% RSLogix 500 project I2P Hands-On 4 - Luke.RSS, saved by version 10.00.00.00 %
PROJECT "UNTITLED"    % processor: Bul.1763 MicroLogix 1100 Series B %

PROGRAM FILES
  LAD 2   13 rungs

DATA FILES
  O0 OUTPUT  4 elements
  I1 INPUT  6 elements
  S2 STATUS  66 elements
  B3 BINARY  1 elements
  T4 TIMER  2 elements
  C5 COUNTER  1 elements
  R6 CONTROL  1 elements
  N7 INTEGER  1 elements
  F8 FLOAT  1 elements

LADDER 2
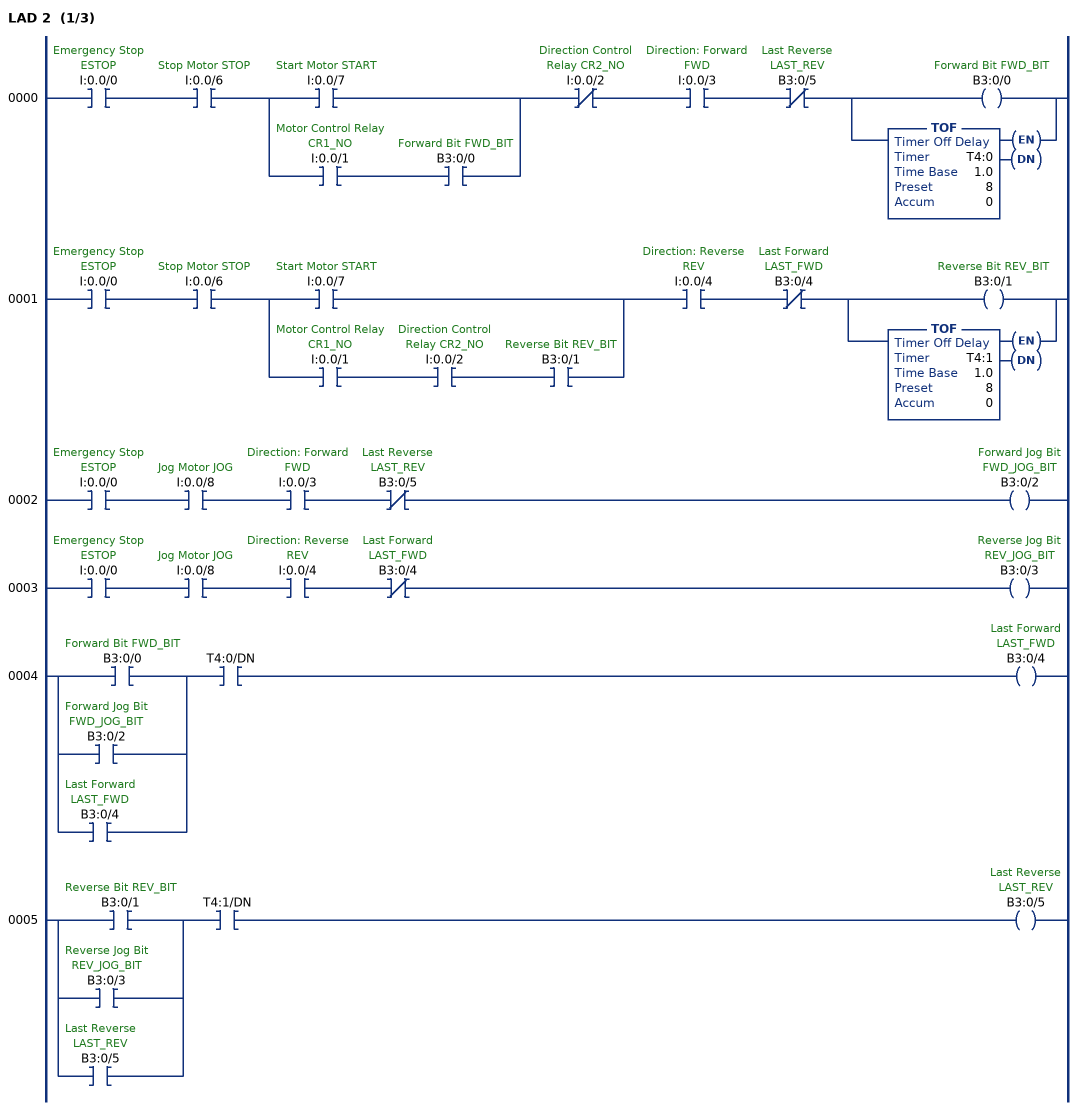
% Rung: 0 %
SOR XIC I:0.0/0 XIC I:0.0/6 BST XIC I:0.0/7 NXB XIC I:0.0/1 XIC B3:0/0 BND XIO I:0.0/2 XIC I:0.0/3 XIO B3:0/5 BST OTE B3:0/0 NXB TOF T4:0 1.0 8 0 BND EOR
%   I:0.0/0  ESTOP  "Emergency Stop" %
%   I:0.0/6  STOP  "Stop Motor" %
%   I:0.0/7  START  "Start Motor" %
%   I:0.0/1  CR1_NO  "Motor Control Relay" %
%   B3:0/0  FWD_BIT  "Forward Bit" %
%   I:0.0/2  CR2_NO  "Direction Control Relay" %
%   I:0.0/3  FWD  "Direction: Forward" %
%   B3:0/5  LAST_REV  "Last Reverse" %
% Rung: 1 %
SOR XIC I:0.0/0 XIC I:0.0/6 BST XIC I:0.0/7 NXB XIC I:0.0/1 XIC I:0.0/2 XIC B3:0/1 BND XIC I:0.0/4 XIO B3:0/4 BST OTE B3:0/1 NXB TOF T4:1 1.0 8 0 BND EOR
%   I:0.0/0  ESTOP  "Emergency Stop" %
%   I:0.0/6  STOP  "Stop Motor" %
%   I:0.0/7  START  "Start Motor" %
%   I:0.0/1  CR1_NO  "Motor Control Relay" %
%   I:0.0/2  CR2_NO  "Direction Control Relay" %
%   B3:0/1  REV_BIT  "Reverse Bit" %
%   I:0.0/4  REV  "Direction: Reverse" %
%   B3:0/4  LAST_FWD  "Last Forward" %
% Rung: 2 %
SOR XIC I:0.0/0 XIC I:0.0/8 XIC I:0.0/3 XIO B3:0/5 OTE B3:0/2 EOR
%   I:0.0/0  ESTOP  "Emergency Stop" %
%   I:0.0/8  JOG  "Jog Motor" %
%   I:0.0/3  FWD  "Direction: Forward" %
%   B3:0/5  LAST_REV  "Last Reverse" %
%   B3:0/2  FWD_JOG_BIT  "Forward Jog Bit" %
% Rung: 3 %
SOR XIC I:0.0/0 XIC I:0.0/8 XIC I:0.0/4 XIO B3:0/4 OTE B3:0/3 EOR
%   I:0.0/0  ESTOP  "Emergency Stop" %
%   I:0.0/8  JOG  "Jog Motor" %
%   I:0.0/4  REV  "Direction: Reverse" %
%   B3:0/4  LAST_FWD  "Last Forward" %
%   B3:0/3  REV_JOG_BIT  "Reverse Jog Bit" %
% Rung: 4 %
SOR BST XIC B3:0/0 NXB BST XIC B3:0/2 NXB XIC B3:0/4 BND BND XIC T4:0/DN OTE B3:0/4 EOR
%   B3:0/0  FWD_BIT  "Forward Bit" %
%   B3:0/2  FWD_JOG_BIT  "Forward Jog Bit" %
%   B3:0/4  LAST_FWD  "Last Forward" %
% Rung: 5 %
SOR BST XIC B3:0/1 NXB BST XIC B3:0/3 NXB XIC B3:0/5 BND BND XIC T4:1/DN OTE B3:0/5 EOR
%   B3:0/1  REV_BIT  "Reverse Bit" %
%   B3:0/3  REV_JOG_BIT  "Reverse Jog Bit" %
%   B3:0/5  LAST_REV  "Last Reverse" %

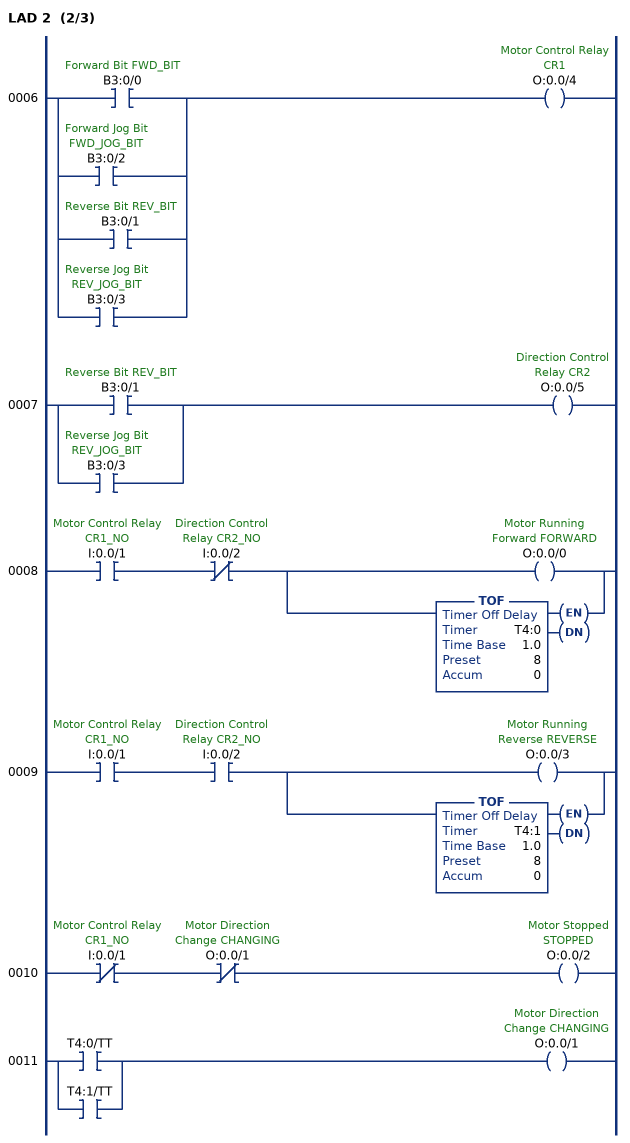
% Rung: 6 %
SOR BST XIC B3:0/0 NXB BST XIC B3:0/2 NXB BST XIC B3:0/1 NXB XIC B3:0/3 BND BND BND OTE O:0.0/4 EOR
%   B3:0/0  FWD_BIT  "Forward Bit" %
%   B3:0/2  FWD_JOG_BIT  "Forward Jog Bit" %
%   B3:0/1  REV_BIT  "Reverse Bit" %
%   B3:0/3  REV_JOG_BIT  "Reverse Jog Bit" %
%   O:0.0/4  CR1  "Motor Control Relay" %
% Rung: 7 %
SOR BST XIC B3:0/1 NXB XIC B3:0/3 BND OTE O:0.0/5 EOR
%   B3:0/1  REV_BIT  "Reverse Bit" %
%   B3:0/3  REV_JOG_BIT  "Reverse Jog Bit" %
%   O:0.0/5  CR2  "Direction Control Relay" %
% Rung: 8 %
SOR XIC I:0.0/1 XIO I:0.0/2 BST OTE O:0.0/0 NXB TOF T4:0 1.0 8 0 BND EOR
%   I:0.0/1  CR1_NO  "Motor Control Relay" %
%   I:0.0/2  CR2_NO  "Direction Control Relay" %
%   O:0.0/0  FORWARD  "Motor Running Forward" %
% Rung: 9 %
SOR XIC I:0.0/1 XIC I:0.0/2 BST OTE O:0.0/3 NXB TOF T4:1 1.0 8 0 BND EOR
%   I:0.0/1  CR1_NO  "Motor Control Relay" %
%   I:0.0/2  CR2_NO  "Direction Control Relay" %
%   O:0.0/3  REVERSE  "Motor Running Reverse" %
% Rung: 10 %
SOR XIO I:0.0/1 XIO O:0.0/1 OTE O:0.0/2 EOR
%   I:0.0/1  CR1_NO  "Motor Control Relay" %
%   O:0.0/1  CHANGING  "Motor Direction Change" %
%   O:0.0/2  STOPPED  "Motor Stopped" %
% Rung: 11 %
SOR BST XIC T4:0/TT NXB XIC T4:1/TT BND OTE O:0.0/1 EOR
%   O:0.0/1  CHANGING  "Motor Direction Change" %

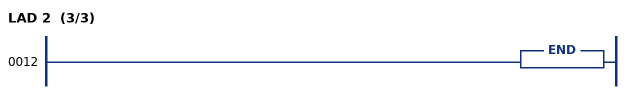
% Rung: 12 %
SOR END EOR

OTHER DOCUMENTED ADDRESSES
  B3:0/6  Y_BIT  "Yellow light bit"
  I:0.0/5  ZZZ  "Direction: Forward- Off-Reverse"

DATA TABLE (non-zero values as saved)
DATA T4
% .PRE .ACC %
% T4:0 % 8 0
% T4:1 % 8 0
